// Mitsubishi GX Works2 project: plc_208837534_316493808   PLC: FX3G

// global labels: Global1
VAR_GLOBAL
  reset AT X010 : BOOL;
  EndDAY AT X005 : BOOL;
  cc17 AT CC17 : BOOL;
END_VAR
VAR_GLOBAL CONSTANT
  k_3 : INT := 3;
END_VAR
VAR_GLOBAL
  startDAY AT CS17 : BOOL;
  LAMP10 AT Y010 : BOOL;
  t_c_1 AT TC1 : BOOL;
END_VAR
VAR_GLOBAL CONSTANT
  k_5 : INT := 500;
END_VAR
VAR_GLOBAL
  LAMP11 AT Y011 : BOOL;
  m_0 AT M0 : BOOL;
END_VAR
VAR_GLOBAL CONSTANT
  k_1 : INT := 2000;
END_VAR
VAR_GLOBAL
  d_110 AT D1100 : INT;
  d_1110 AT D1110 : INT;
END_VAR
VAR_GLOBAL CONSTANT
  k_500 : INT := 50;
END_VAR
VAR_GLOBAL
  m_1 AT M1 : BOOL;
  t_c_3 AT TC3 : BOOL;
END_VAR
VAR_GLOBAL CONSTANT
  k_50 : INT := 50;
END_VAR
VAR_GLOBAL
  t_n_3 AT TN3 : INT;
  t_s_3 AT TS3 : BOOL;
END_VAR
VAR_GLOBAL CONSTANT
  Processing : REAL := 1350;
  Coating : REAL := 4500;
END_VAR
VAR_GLOBAL
  chocolate AT D1125 : REAL;
  StartOfProcessing AT X001 : BOOL;
  PeanutProcessing AT D1130 : REAL;
END_VAR
VAR_GLOBAL CONSTANT
  MAX150 : REAL := 150;
END_VAR
VAR_GLOBAL
  Peanut AT D1120 : REAL;
  HELP AT D1103 : INT;
  M_3 AT M3 : BOOL;
  m_4 AT M4 : BOOL;
  m_5 AT M5 : BOOL;
  LessThen70 AT M5 : BOOL;
  LessThen120 AT M6 : BOOL;
  LessThen150 AT M7 : BOOL;
END_VAR
VAR_GLOBAL CONSTANT
  k_120 : REAL := 120;
  k_150 : REAL := 150;
  k_70 : REAL := 70;
  k_20 : INT := 20;
  k_30 : INT := 30;
  k_40 : INT := 40;
END_VAR
VAR_GLOBAL
  m_8 AT M8 : BOOL;
  lampy1 AT Y001 : BOOL;
  d_1112 AT D1112 : INT;
  d_1114 AT D1114 : INT;
  d_1118 AT D1118 : INT;
  t_c_2 AT TC2 : BOOL;
  t_c_4 AT TC4 : BOOL;
  t_s_2 AT TS2 : BOOL;
  t_n_2 AT TN2 : INT;
  t_s_1 AT TS1 : BOOL;
  t_s_4 AT TS4 : BOOL;
  t_n_4 AT TN4 : INT;
END_VAR
VAR_GLOBAL CONSTANT
  k_45 : INT := 45;
  k_60 : INT := 60;
END_VAR
VAR_GLOBAL
  t_c_5 AT TC5 : BOOL;
  t_c_6 AT TC6 : BOOL;
  t_c_7 AT TC7 : BOOL;
  t_s_5 AT TS5 : BOOL;
  t_s_6 AT TS6 : BOOL;
  t_s_7 AT TS7 : BOOL;
  t_c_8 AT TC8 : BOOL;
  m_11 AT M11 : BOOL;
  t_s_8 AT TS8 : BOOL;
  t_c_9 AT TC9 : BOOL;
  t_s_9 AT TS9 : BOOL;
  LAMP3 AT Y003 : BOOL;
  t_c_10 AT TC10 : BOOL;
END_VAR
VAR_GLOBAL CONSTANT
  k_10 : INT := 10;
END_VAR
VAR_GLOBAL
  t_s_10 AT TS10 : BOOL;
  t_c_11 AT TC11 : BOOL;
  t_s_11 AT TS11 : BOOL;
  m_12 AT M12 : BOOL;
  t_n_10 AT TN10 : INT;
END_VAR
VAR_GLOBAL CONSTANT
  k_100 : INT := 100;
END_VAR
VAR_GLOBAL
  t_c_15 AT TC15 : BOOL;
  t_s_15 AT TS15 : BOOL;
  t_c_20 AT TC20 : BOOL;
  t_s_20 AT TS20 : BOOL;
  m_13 AT M13 : BOOL;
  t_c_25 AT TC25 : BOOL;
  t_s_25 AT TS25 : BOOL;
  t_n_25 AT TN25 : INT;
  t_n_15 AT TN15 : INT;
  d_1160 AT D1160 : INT;
  t_c_30 AT TC30 : BOOL;
  m_14 AT M14 : BOOL;
  t_s_30 AT TS30 : BOOL;
  m_15 AT M15 : BOOL;
  m_16 AT M16 : BOOL;
  m_17 AT M17 : BOOL;
END_VAR
VAR_GLOBAL CONSTANT
  MAX600chocolate : REAL := 600;
END_VAR
VAR_GLOBAL
  m_18 AT M18 : BOOL;
  readAnalog AT X007 : BOOL;
END_VAR
VAR_GLOBAL CONSTANT
  k_2_5 : REAL := 2.5;
  k_7 : REAL := 7;
END_VAR
VAR_GLOBAL
  m_19 AT M19 : BOOL;
END_VAR
VAR_GLOBAL CONSTANT
  k_9 : REAL := 9;
END_VAR
VAR_GLOBAL
  m_20 AT M20 : BOOL;
END_VAR
VAR_GLOBAL CONSTANT
  k_1_1 : REAL := 1;
END_VAR
VAR_GLOBAL
  m_21 AT M21 : BOOL;
  m_22 AT M22 : BOOL;
  m_23 AT M23 : BOOL;
  EndTransformationProcess AT M9 : BOOL;
  EndCuttingProcess AT M10 : BOOL;
END_VAR
VAR_GLOBAL CONSTANT
  k_0 : REAL;
END_VAR
VAR_GLOBAL
  analogIn2 AT D8281 : INT;
  valueBamba AT D1145 : REAL;
  d_1170 AT D1170 : INT;
END_VAR
VAR_GLOBAL CONSTANT
  K_397_2 : REAL := 397.2;
END_VAR
VAR_GLOBAL
  valueBambaGOOD AT D1150 : REAL;
  m_24 AT M24 : BOOL;
  EndValue AT M25 : BOOL;
END_VAR
VAR_GLOBAL CONSTANT
  k_1_5 : REAL := 1.5;
END_VAR
VAR_GLOBAL
  c_o AT M26 : BOOL;
  x_2 AT X002 : BOOL;
  x_3 AT X003 : BOOL;
  Coating_container AT D1135 : REAL;
  THERE_IS_CHOCOLATE AT M27 : BOOL;
  amountProsecs AT D1105 : REAL;
END_VAR
VAR_GLOBAL CONSTANT
  k_3_3 : REAL := 3;
END_VAR
VAR_GLOBAL
  m_28 AT M28 : BOOL;
  m_29 AT M29 : BOOL;
  time_Coating AT D1165 : INT;
END_VAR
VAR_GLOBAL CONSTANT
  k_4 : INT := 4;
  k_5_5 : INT := 50;
END_VAR
VAR_GLOBAL
  M_30 AT M30 : BOOL;
  t_c_40 AT TC40 : BOOL;
  t_s_40 AT TS40 : BOOL;
  t_c_45 AT TC45 : BOOL;
  t_s_45 AT TS45 : BOOL;
  y_6 AT Y006 : BOOL;
  t_c_50 AT TC50 : BOOL;
  t_s_50 AT TS50 : BOOL;
  M_31 AT M31 : BOOL;
END_VAR
VAR_GLOBAL CONSTANT
  k_2 : REAL := 2;
END_VAR
VAR_GLOBAL
  Bamba_bags AT D1175 : REAL;
  m_32 AT M32 : BOOL;
  Bamba_bags_int AT D1180 : INT;
  M_33 AT M33 : BOOL;
  M_34 AT M34 : BOOL;
  M_35 AT M35 : BOOL;
  M_36 AT M36 : BOOL;
END_VAR
VAR_GLOBAL CONSTANT
  k_50_0 : INT := 500;
END_VAR
VAR_GLOBAL
  M_37 AT M37 : BOOL;
END_VAR
VAR_GLOBAL CONSTANT
  k_5000 : INT := 5000;
END_VAR
VAR_GLOBAL
  M_38 AT M38 : BOOL;
  M_39 AT M39 : BOOL;
END_VAR
VAR_GLOBAL CONSTANT
  k_10_10 : INT := 10;
END_VAR
VAR_GLOBAL
  amout_Contenirs_to_int AT D1195 : INT;
  Bags AT D1185 : INT;
  Amount_Contenirs AT D1190 : INT;
  m_40 AT M40 : BOOL;
  modolu AT D1200 : INT;
  m_41 AT M41 : BOOL;
END_VAR
VAR_GLOBAL CONSTANT
  k_1_word : INT := 1;
END_VAR
VAR_GLOBAL
  m_42 AT M42 : BOOL;
END_VAR
VAR_GLOBAL CONSTANT
  k_0_0 : INT;
END_VAR
VAR_GLOBAL
  m_43 AT M43 : BOOL;
  Container_after_work_cot AT M44 : BOOL;
  Container_after_work_pean AT M45 : BOOL;
END_VAR
VAR_GLOBAL CONSTANT
  k_2500 : INT := 2500;
END_VAR
VAR_GLOBAL
  five_ton AT M46 : BOOL;
  t_c_70 AT TC70 : BOOL;
  t_s_70 AT TS70 : BOOL;
  lampy7 AT Y007 : BOOL;
  m_50 AT M50 : BOOL;
END_VAR
VAR_GLOBAL CONSTANT
  k_0_1 : REAL := 0.1;
END_VAR
VAR_GLOBAL
  there_is_peant AT M47 : BOOL;
  No_storage_space_END_DAY AT M49 : BOOL;
  Completion_coating_proces AT M51 : BOOL;
  Out_chocolate_stock AT M52 : BOOL;
  Out_peanut_stok AT M53 : BOOL;
  Conditions_ending_day AT M54 : BOOL;
END_VAR
VAR_GLOBAL CONSTANT
  k_2_WORD : INT := 2;
END_VAR
VAR_GLOBAL
  Duplication_performed AT M55 : BOOL;
END_VAR
VAR_GLOBAL CONSTANT
  k_1000 : REAL := 1000;
END_VAR
VAR_GLOBAL
  Distribution_made AT M56 : BOOL;
  Div_made AT M57 : BOOL;
  reset_variables AT M58 : BOOL;
END_VAR
VAR_GLOBAL CONSTANT
  K_397_2_WORD : INT := 397;
END_VAR
VAR_GLOBAL
  Several_processes AT CC20 : BOOL;
  cS20 AT CS20 : BOOL;
  bags_in_float AT D1240 : REAL;
  bamba_to_float AT M60 : BOOL;
  Amount_bamba_kg AT D1210 : REAL;
  Amount_bamba_ton AT D1220 : REAL;
  Amouny_bamba_analog AT D1230 : REAL;
  Bamab_output AT D1250 : INT;
  move_to_int AT M61 : BOOL;
  analog_output AT D8282 : INT;
  print_to_analog AT M62 : BOOL;
END_VAR
VAR_GLOBAL CONSTANT
  k_2_6 : REAL := 2.6;
  k_7_1 : REAL := 7.1;
  k_70_1 : REAL := 70.1;
  k_120_1 : REAL := 120.1;
END_VAR
VAR_GLOBAL
  M_63 AT M63 : BOOL;
END_VAR

// task Task_01 (event TRUE, interval 0, priority 31): POU_01

PROGRAM POU_01
(* structured ladder/FBD written out as ST: instructions are called as NAME(EN, inputs, outputs); _pN, _eN, _tN stand for wires *)
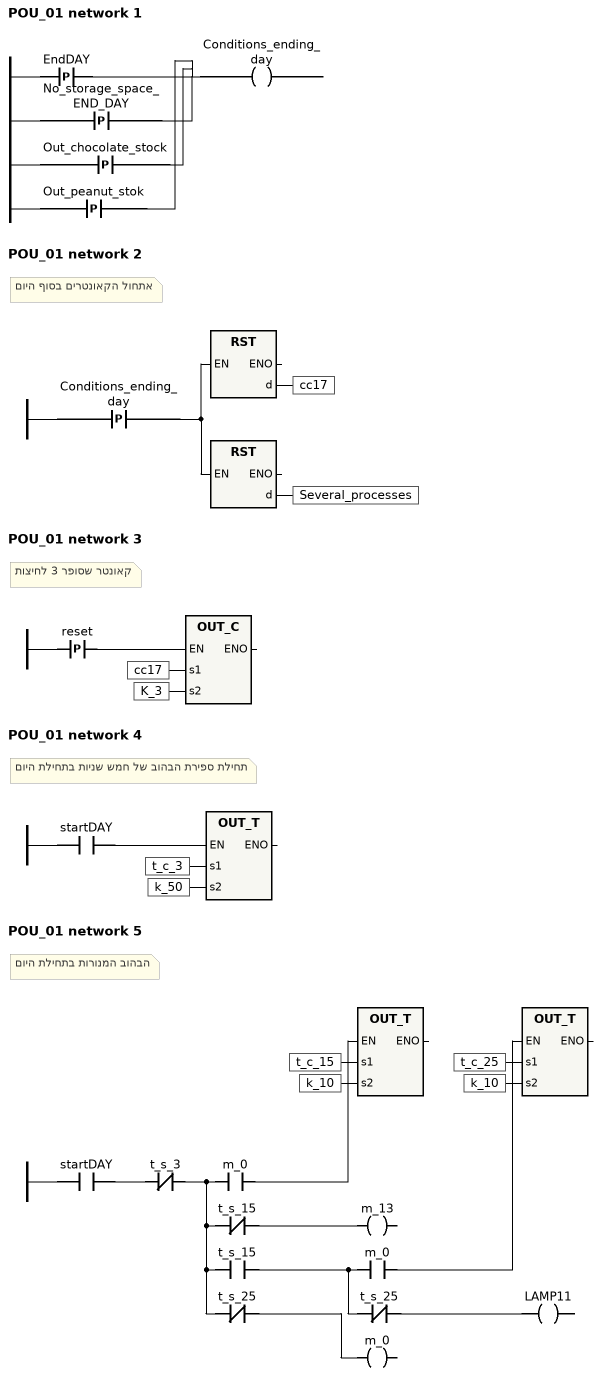
(* network 1 *)
Conditions_ending_day := LDP(TRUE, EndDAY) OR LDP(TRUE, No_storage_space_END_DAY) OR LDP(TRUE, Out_chocolate_stock) OR LDP(TRUE, Out_peanut_stok);
(* network 2 *)
(* אתחול הקאונטרים בסוף היום *)
_p1 := LDP(TRUE, Conditions_ending_day);
RST(_p1, cc17);
RST(_p1, Several_processes);
(* network 3 *)
(* קאונטר שסופר 3 לחיצות *)
OUT_C(LDP(TRUE, reset), cc17, K_3);
(* network 4 *)
(* תחילת ספירת הבהוב של חמש שניות בתחילת היום *)
OUT_T(startDAY, t_c_3, k_50);
(* network 5 *)
(* הבהוב המנורות בתחילת היום *)
_p1 := startDAY AND NOT t_s_3;
OUT_T(_p1 AND m_0, t_c_15, k_10);
m_13 := _p1 AND NOT t_s_15;
_p2 := _p1 AND t_s_15;
OUT_T(_p2 AND m_0, t_c_25, k_10);
LAMP11 := _p2 AND NOT t_s_25;
m_0 := _p1 AND NOT t_s_25;
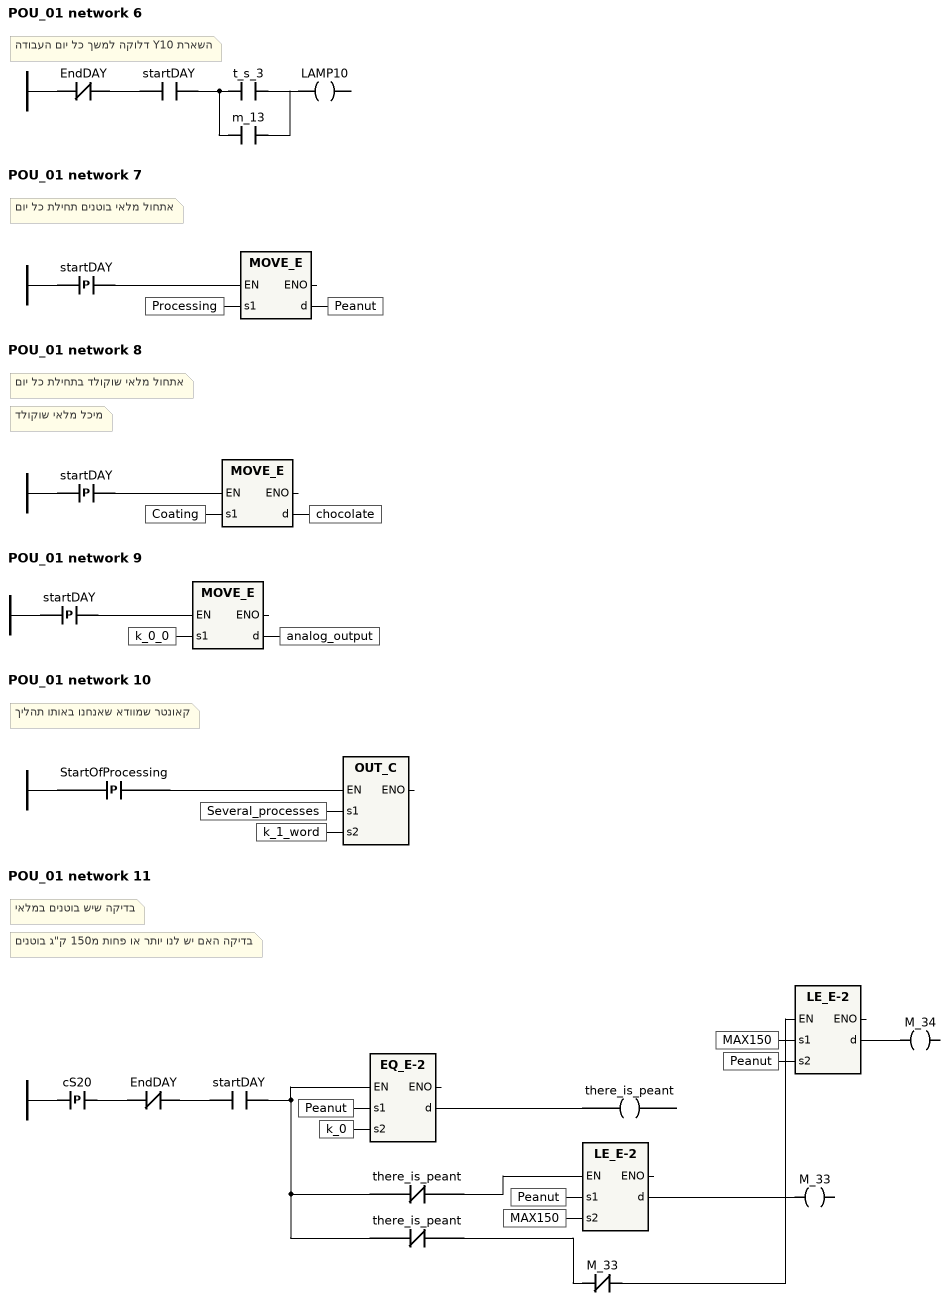
(* network 6 *)
(* השארת Y10 דלוקה למשך כל יום העבודה *)
_p1 := NOT EndDAY AND startDAY;
LAMP10 := (_p1 AND t_s_3) OR (_p1 AND m_13);
(* network 7 *)
(* אתחול מלאי בוטנים תחילת כל יום *)
MOVE_E(LDP(TRUE, startDAY), Processing, Peanut);
(* network 8 *)
(* אתחול מלאי שוקולד בתחילת כל יום *)
(* מיכל מלאי שוקולד *)
MOVE_E(LDP(TRUE, startDAY), Coating, chocolate);
(* network 9 *)
MOVE_E(LDP(TRUE, startDAY), k_0_0, analog_output);
(* network 10 *)
(* קאונטר שמוודא שאנחנו באותו תהליך *)
OUT_C(LDP(TRUE, StartOfProcessing), Several_processes, k_1_word);
(* network 11 *)
(* בדיקה שיש בוטנים במלאי *)
(* בדיקה האם יש לנו יותר או פחות מ150 ק"ג בוטנים *)
_p1 := LDP(TRUE, cS20) AND NOT EndDAY AND startDAY;
EQ_E(_p1, Peanut, k_0, _t2);
there_is_peant := _t2;
LE_E(_p1 AND NOT there_is_peant, Peanut, MAX150, _t3);
M_33 := _t3;
LE_E(_p1 AND NOT there_is_peant AND NOT M_33, MAX150, Peanut, _t4);
M_34 := _t4;
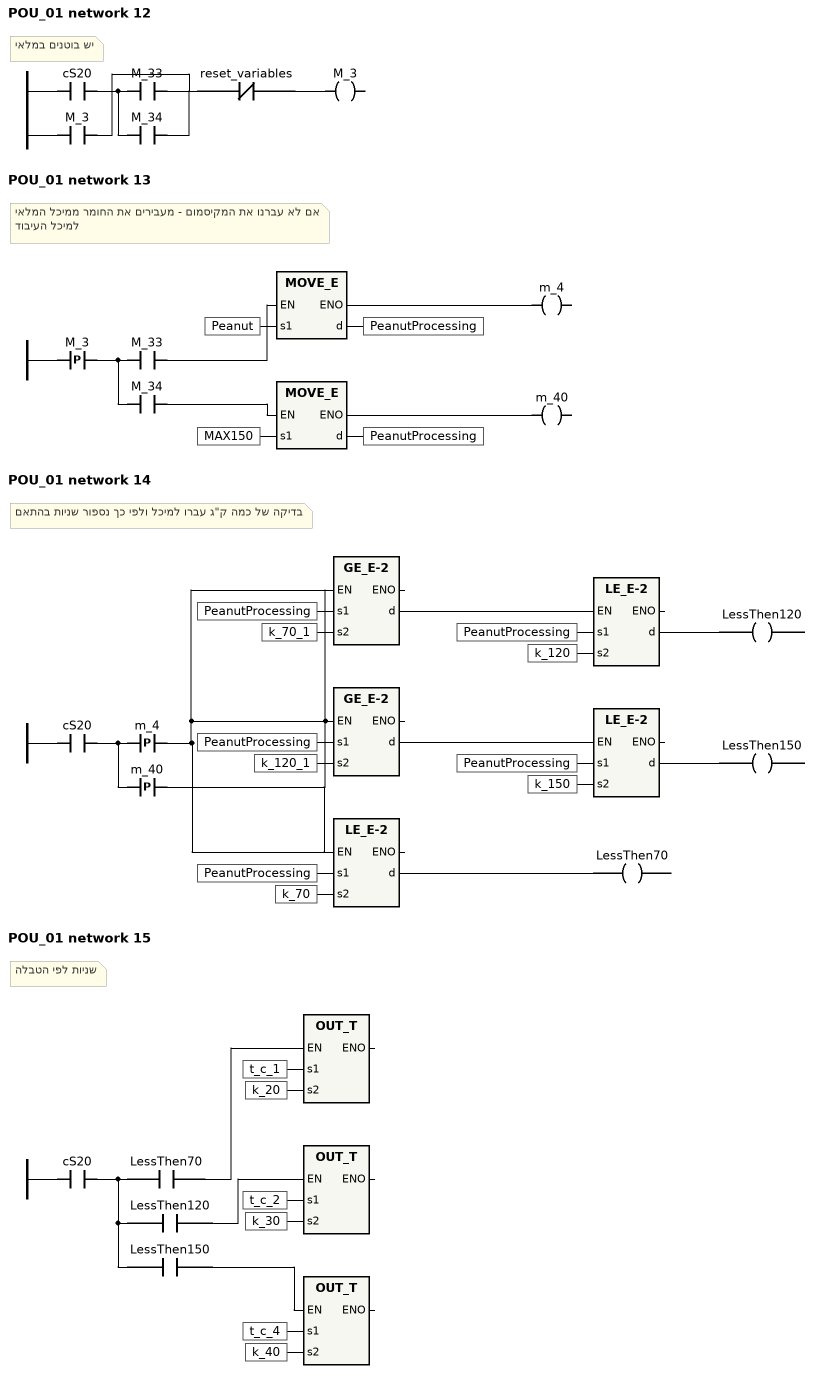
(* network 12 *)
(* יש בוטנים במלאי *)
M_3 := ((cS20 AND M_33) OR (cS20 AND M_34) OR M_3) AND NOT reset_variables;
(* network 13 *)
(* אם לא עברנו את המקיסמום - מעבירים את החומר ממיכל המלאי למיכל העיבוד *)
_p1 := LDP(TRUE, M_3);
_e2 := MOVE_E(_p1 AND M_33, Peanut, PeanutProcessing);
m_4 := _e2;
_e3 := MOVE_E(_p1 AND M_34, MAX150, PeanutProcessing);
m_40 := _e3;
(* network 14 *)
(* בדיקה של כמה ק"ג עברו למיכל ולפי כך נספור שניות בהתאם *)
_p1 := (cS20 AND LDP(TRUE, m_4)) OR (cS20 AND LDP(TRUE, m_40));
LE_E(_p1, PeanutProcessing, k_70, _t2);
LessThen70 := _t2;
GE_E(_p1, PeanutProcessing, k_70_1, _t3);
LE_E(_t3, PeanutProcessing, k_120, _t4);
LessThen120 := _t4;
GE_E(_p1, PeanutProcessing, k_120_1, _t5);
LE_E(_t5, PeanutProcessing, k_150, _t6);
LessThen150 := _t6;
(* network 15 *)
(* שניות לפי הטבלה *)
OUT_T(cS20 AND LessThen70, t_c_1, k_20);
OUT_T(cS20 AND LessThen120, t_c_2, k_30);
OUT_T(cS20 AND LessThen150, t_c_4, k_40);
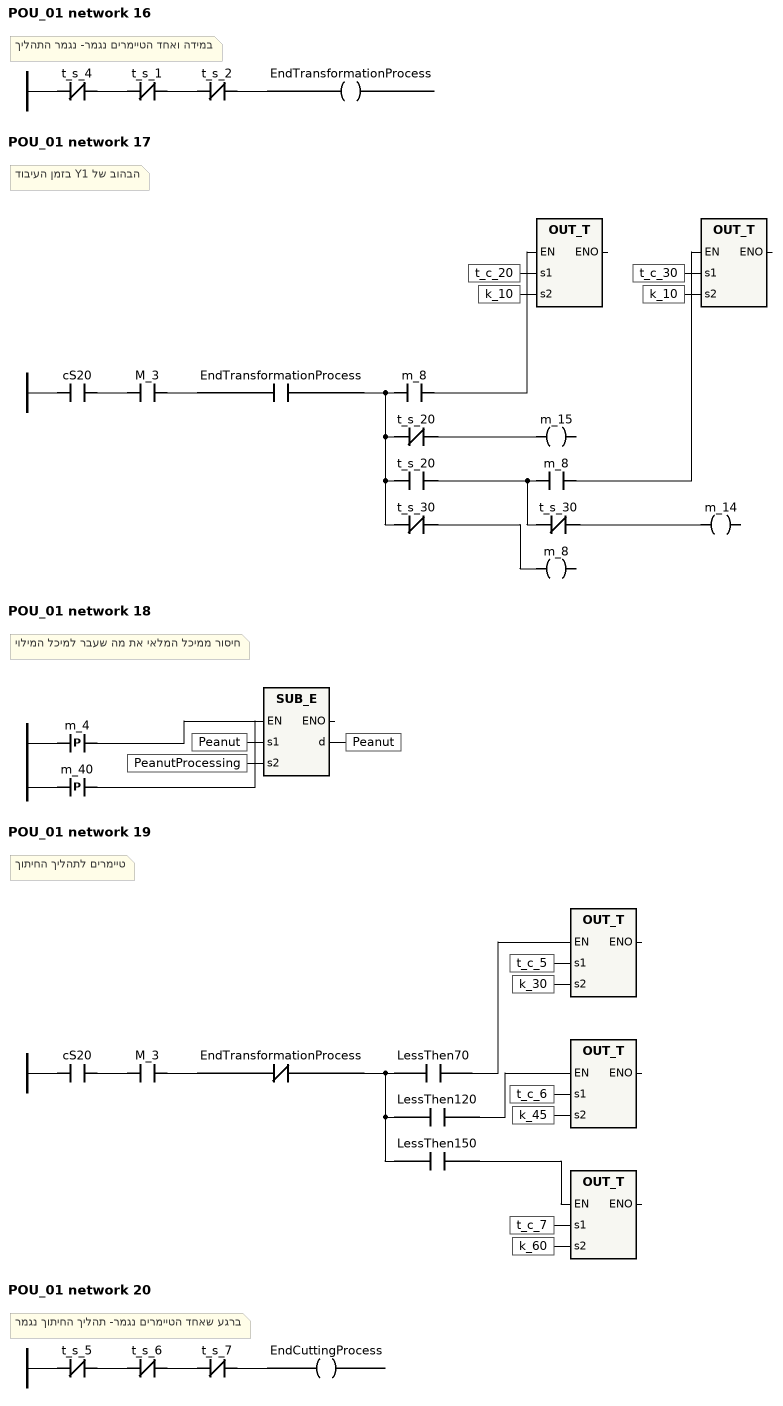
(* network 16 *)
(* במידה ואחד הטיימרים נגמר- נגמר התהליך *)
EndTransformationProcess := NOT t_s_4 AND NOT t_s_1 AND NOT t_s_2;
(* network 17 *)
(* הבהוב של Y1 בזמן העיבוד *)
_p1 := cS20 AND M_3 AND EndTransformationProcess;
OUT_T(_p1 AND m_8, t_c_20, k_10);
m_15 := _p1 AND NOT t_s_20;
_p2 := _p1 AND t_s_20;
OUT_T(_p2 AND m_8, t_c_30, k_10);
m_14 := _p2 AND NOT t_s_30;
m_8 := _p1 AND NOT t_s_30;
(* network 18 *)
(* חיסור ממיכל המלאי את מה שעבר למיכל המילוי *)
SUB_E(LDP(TRUE, m_4) OR LDP(TRUE, m_40), Peanut, PeanutProcessing, Peanut);
(* network 19 *)
(* טיימרים לתהליך החיתוך *)
_p1 := cS20 AND M_3 AND NOT EndTransformationProcess;
OUT_T(_p1 AND LessThen70, t_c_5, k_30);
OUT_T(_p1 AND LessThen120, t_c_6, k_45);
OUT_T(_p1 AND LessThen150, t_c_7, k_60);
(* network 20 *)
(* ברגע שאחד הטיימרים נגמר- תהליך החיתוך נגמר *)
EndCuttingProcess := NOT t_s_5 AND NOT t_s_6 AND NOT t_s_7;
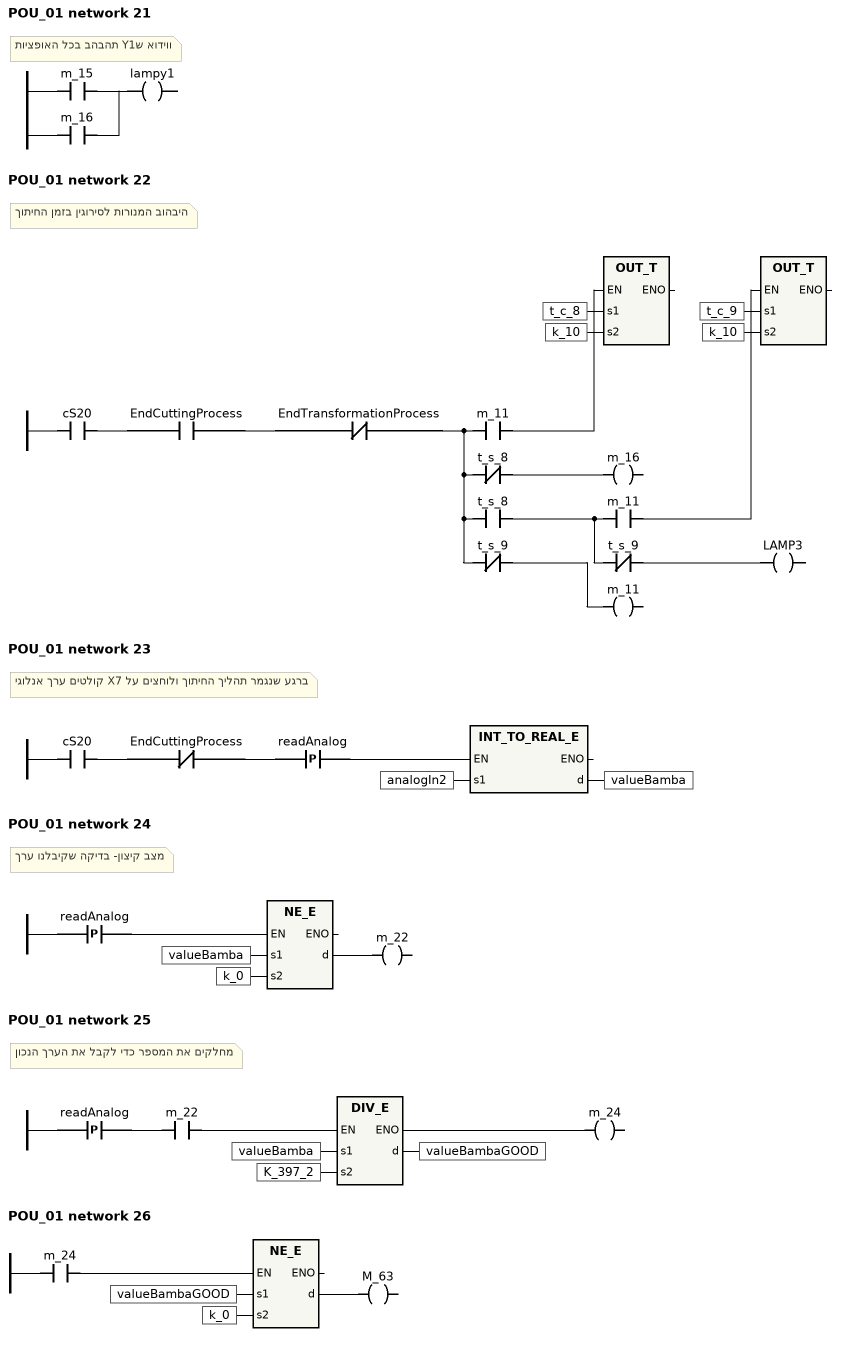
(* network 21 *)
(* ווידוא שY1 תהבהב בכל האופציות *)
lampy1 := m_15 OR m_16;
(* network 22 *)
(* היבהוב המנורות לסירוגין בזמן החיתוך *)
_p1 := cS20 AND EndCuttingProcess AND NOT EndTransformationProcess;
OUT_T(_p1 AND m_11, t_c_8, k_10);
m_16 := _p1 AND NOT t_s_8;
_p2 := _p1 AND t_s_8;
OUT_T(_p2 AND m_11, t_c_9, k_10);
LAMP3 := _p2 AND NOT t_s_9;
m_11 := _p1 AND NOT t_s_9;
(* network 23 *)
(* ברגע שנגמר תהליך החיתוך ולוחצים על X7 קולטים ערך אנלוגי *)
INT_TO_REAL_E(cS20 AND NOT EndCuttingProcess AND LDP(TRUE, readAnalog), analogIn2, valueBamba);
(* network 24 *)
(* מצב קיצון- בדיקה שקיבלנו ערך *)
NE_E(LDP(TRUE, readAnalog), valueBamba, k_0, _t1);
m_22 := _t1;
(* network 25 *)
(* מחלקים את המספר כדי לקבל את הערך הנכון *)
_e1 := DIV_E(LDP(TRUE, readAnalog) AND m_22, valueBamba, K_397_2, valueBambaGOOD);
m_24 := _e1;
(* network 26 *)
NE_E(m_24, valueBambaGOOD, k_0, _t1);
M_63 := _t1;
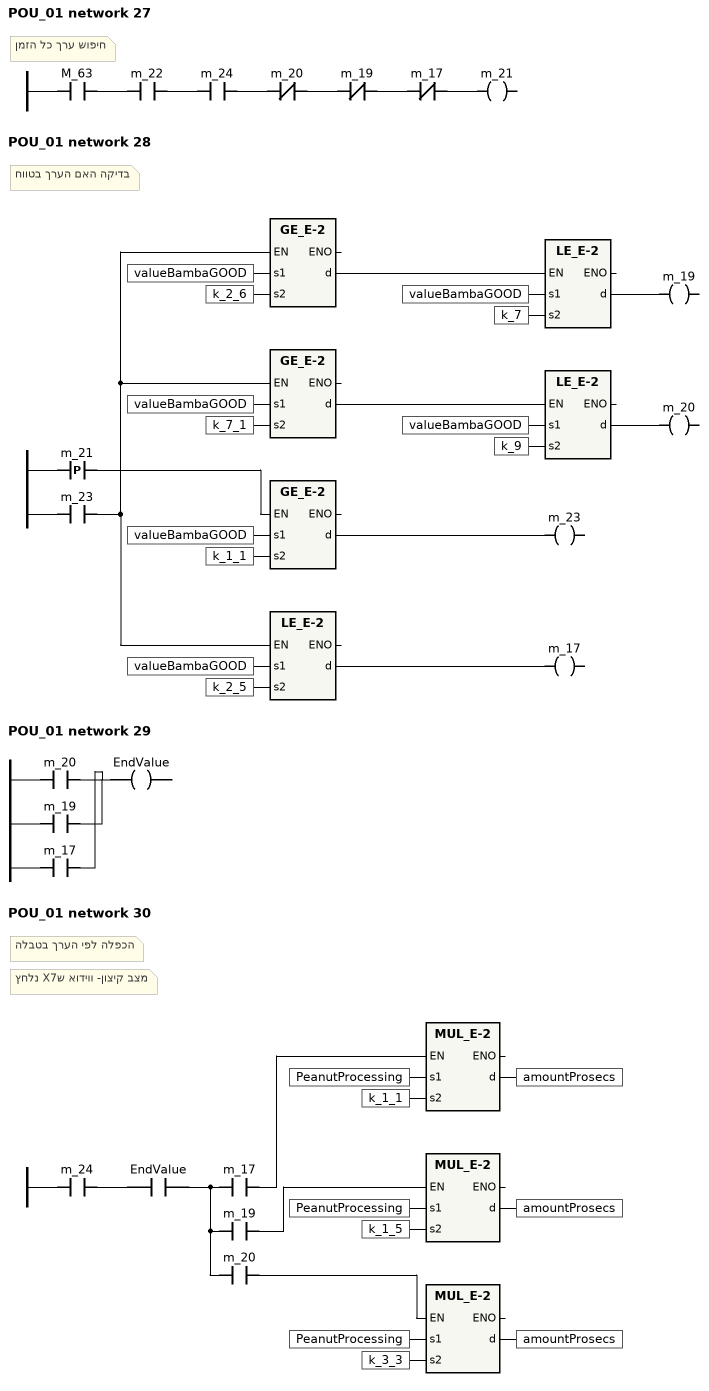
(* network 27 *)
(* חיפוש ערך כל הזמן *)
m_21 := M_63 AND m_22 AND m_24 AND NOT m_20 AND NOT m_19 AND NOT m_17;
(* network 28 *)
(* בדיקה האם הערך בטווח *)
GE_E(LDP(TRUE, m_21), valueBambaGOOD, k_1_1, _t1);
m_23 := _t1;
LE_E(m_23, valueBambaGOOD, k_2_5, _t2);
m_17 := _t2;
GE_E(m_23, valueBambaGOOD, k_2_6, _t3);
LE_E(_t3, valueBambaGOOD, k_7, _t4);
m_19 := _t4;
GE_E(m_23, valueBambaGOOD, k_7_1, _t5);
LE_E(_t5, valueBambaGOOD, k_9, _t6);
m_20 := _t6;
(* network 29 *)
EndValue := m_20 OR m_19 OR m_17;
(* network 30 *)
(* הכפלה לפי הערך בטבלה *)
(* מצב קיצון- ווידוא שX7 נלחץ *)
_p1 := m_24 AND EndValue;
MUL_E(_p1 AND m_17, PeanutProcessing, k_1_1, amountProsecs);
MUL_E(_p1 AND m_19, PeanutProcessing, k_1_5, amountProsecs);
MUL_E(_p1 AND m_20, PeanutProcessing, k_3_3, amountProsecs);
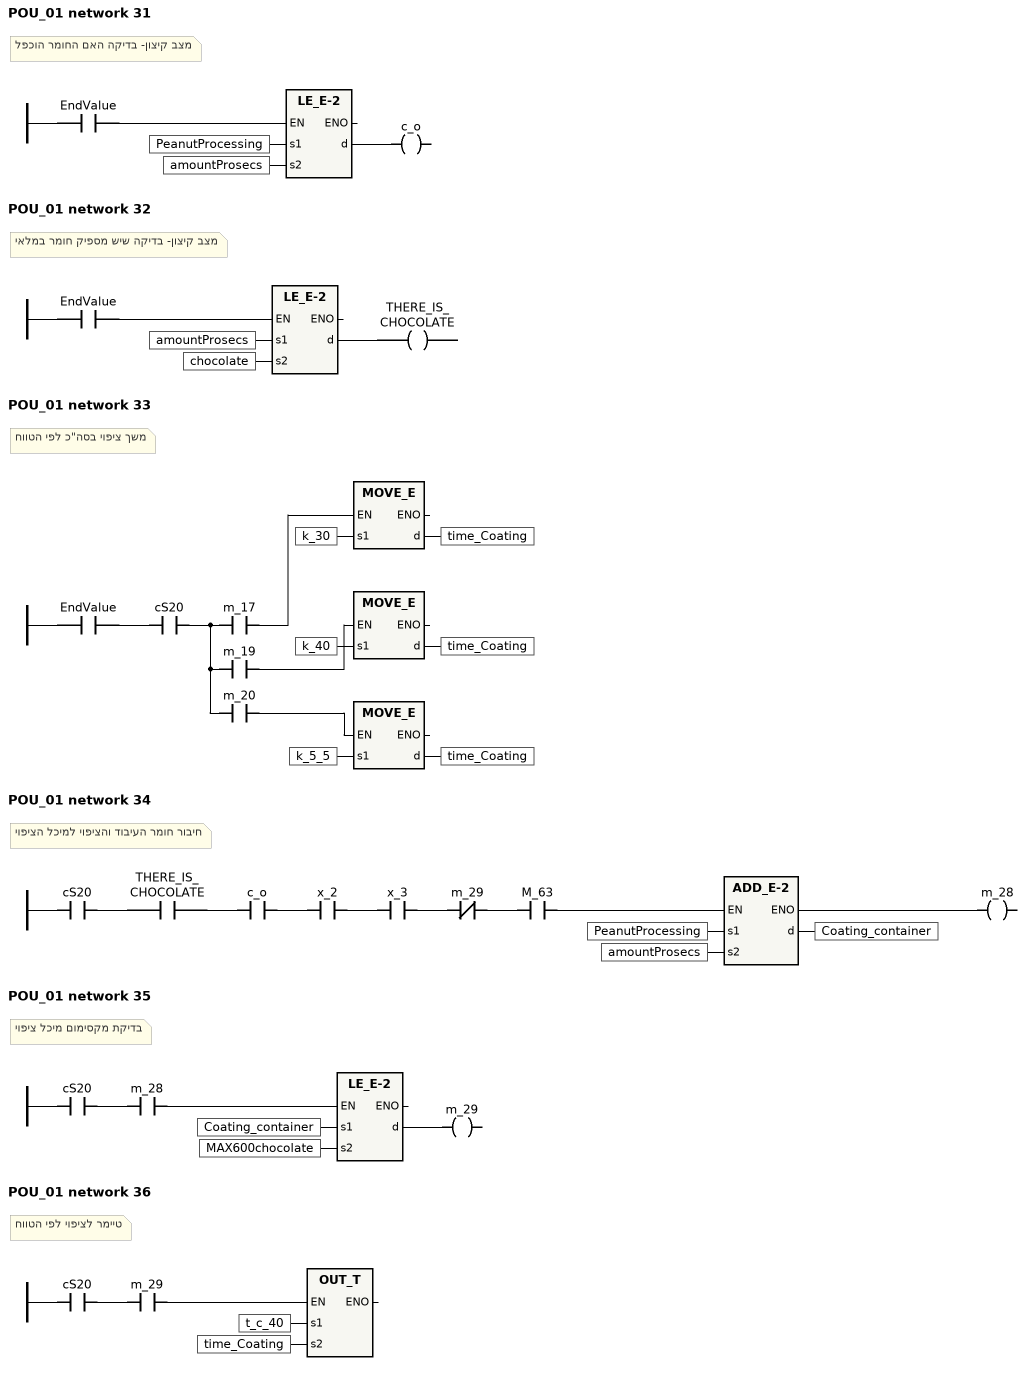
(* network 31 *)
(* מצב קיצון- בדיקה האם החומר הוכפל *)
LE_E(EndValue, PeanutProcessing, amountProsecs, _t1);
c_o := _t1;
(* network 32 *)
(* מצב קיצון- בדיקה שיש מספיק חומר במלאי *)
LE_E(EndValue, amountProsecs, chocolate, _t1);
THERE_IS_CHOCOLATE := _t1;
(* network 33 *)
(* משך ציפוי בסה"כ לפי הטווח *)
_p1 := EndValue AND cS20;
MOVE_E(_p1 AND m_17, k_30, time_Coating);
MOVE_E(_p1 AND m_19, k_40, time_Coating);
MOVE_E(_p1 AND m_20, k_5_5, time_Coating);
(* network 34 *)
(* חיבור חומר העיבוד והציפוי למיכל הציפוי *)
_e1 := ADD_E(cS20 AND THERE_IS_CHOCOLATE AND c_o AND x_2 AND x_3 AND NOT m_29 AND M_63, PeanutProcessing, amountProsecs, Coating_container);
m_28 := _e1;
(* network 35 *)
(* בדיקת מקסימום מיכל ציפוי *)
LE_E(cS20 AND m_28, Coating_container, MAX600chocolate, _t1);
m_29 := _t1;
(* network 36 *)
(* טיימר לציפוי לפי הטווח *)
OUT_T(cS20 AND m_29, t_c_40, time_Coating);
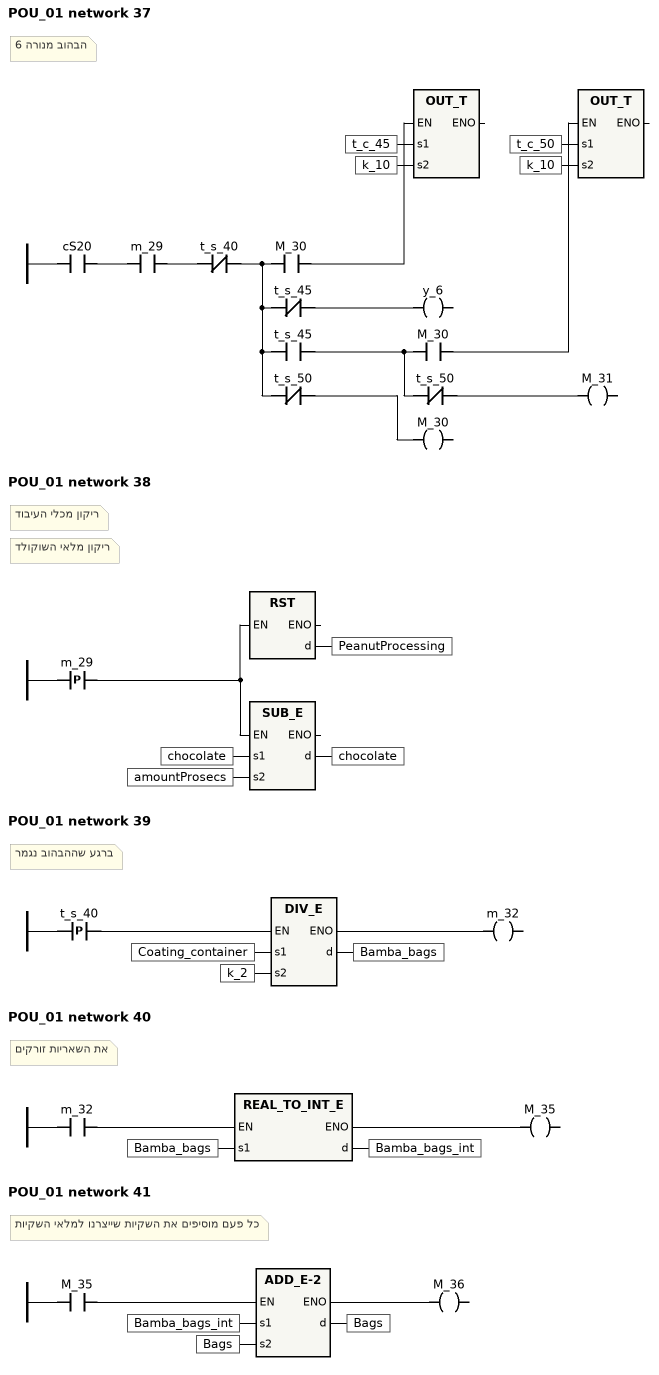
(* network 37 *)
(* הבהוב מנורה 6 *)
_p1 := cS20 AND m_29 AND NOT t_s_40;
OUT_T(_p1 AND M_30, t_c_45, k_10);
y_6 := _p1 AND NOT t_s_45;
_p2 := _p1 AND t_s_45;
OUT_T(_p2 AND M_30, t_c_50, k_10);
M_31 := _p2 AND NOT t_s_50;
M_30 := _p1 AND NOT t_s_50;
(* network 38 *)
(* ריקון מכלי העיבוד *)
(* ריקון מלאי השוקולד *)
_p1 := LDP(TRUE, m_29);
RST(_p1, PeanutProcessing);
SUB_E(_p1, chocolate, amountProsecs, chocolate);
(* network 39 *)
(* ברגע שההבהוב נגמר *)
_e1 := DIV_E(LDP(TRUE, t_s_40), Coating_container, k_2, Bamba_bags);
m_32 := _e1;
(* network 40 *)
(* את השאריות זורקים *)
_e1 := REAL_TO_INT_E(m_32, Bamba_bags, Bamba_bags_int);
M_35 := _e1;
(* network 41 *)
(* כל פעם מוסיפים את השקיות שייצרנו למלאי השקיות *)
_e1 := ADD_E(M_35, Bamba_bags_int, Bags, Bags);
M_36 := _e1;
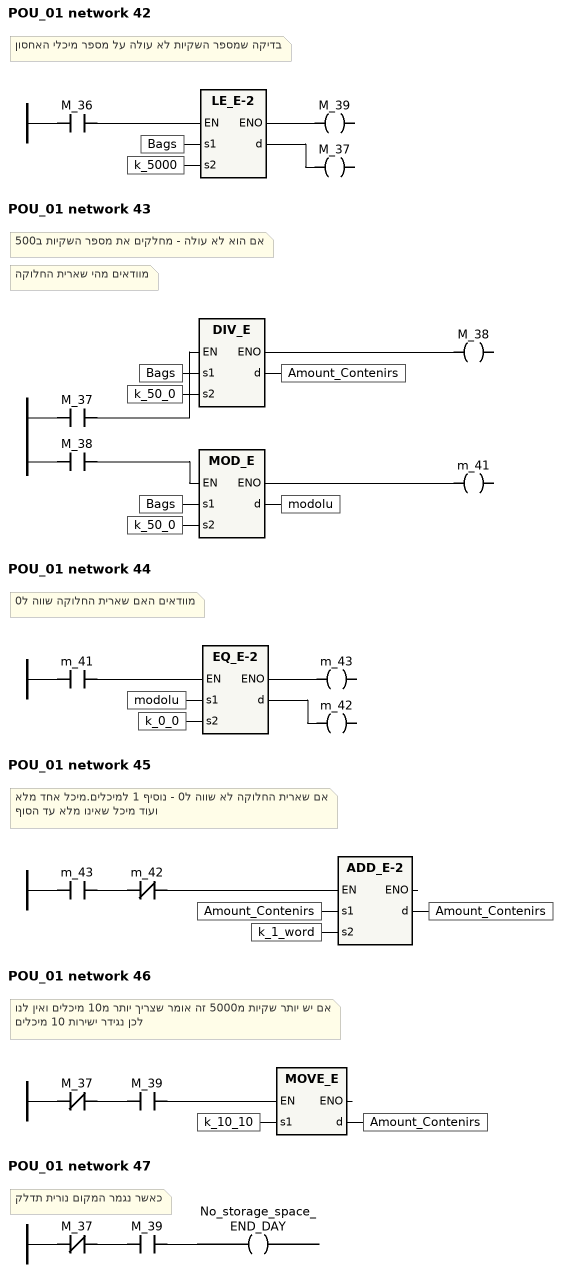
(* network 42 *)
(* בדיקה שמספר השקיות לא עולה על מספר מיכלי האחסון *)
_e2 := LE_E(M_36, Bags, k_5000, _t1);
M_39 := _e2;
M_37 := _t1;
(* network 43 *)
(* אם הוא לא עולה - מחלקים את מספר השקיות ב500 *)
(* מוודאים מהי שארית החלוקה *)
_e1 := DIV_E(M_37, Bags, k_50_0, Amount_Contenirs);
M_38 := _e1;
_e2 := MOD_E(M_38, Bags, k_50_0, modolu);
m_41 := _e2;
(* network 44 *)
(* מוודאים האם שארית החלוקה שווה ל0 *)
_e2 := EQ_E(m_41, modolu, k_0_0, _t1);
m_43 := _e2;
m_42 := _t1;
(* network 45 *)
(* אם שארית החלוקה לא שווה ל0 - נוסיף 1 למיכלים.מיכל אחד מלא ועוד מיכל שאינו מלא עד הסוף *)
ADD_E(m_43 AND NOT m_42, Amount_Contenirs, k_1_word, Amount_Contenirs);
(* network 46 *)
(* אם יש יותר שקיות מ5000 זה אומר שצריך יותר מ10 מיכלים ואין לנו לכן נגידר ישירות 10 מיכלים *)
MOVE_E(NOT M_37 AND M_39, k_10_10, Amount_Contenirs);
(* network 47 *)
(* כאשר נגמר המקום נורית תדלק *)
No_storage_space_END_DAY := NOT M_37 AND M_39;
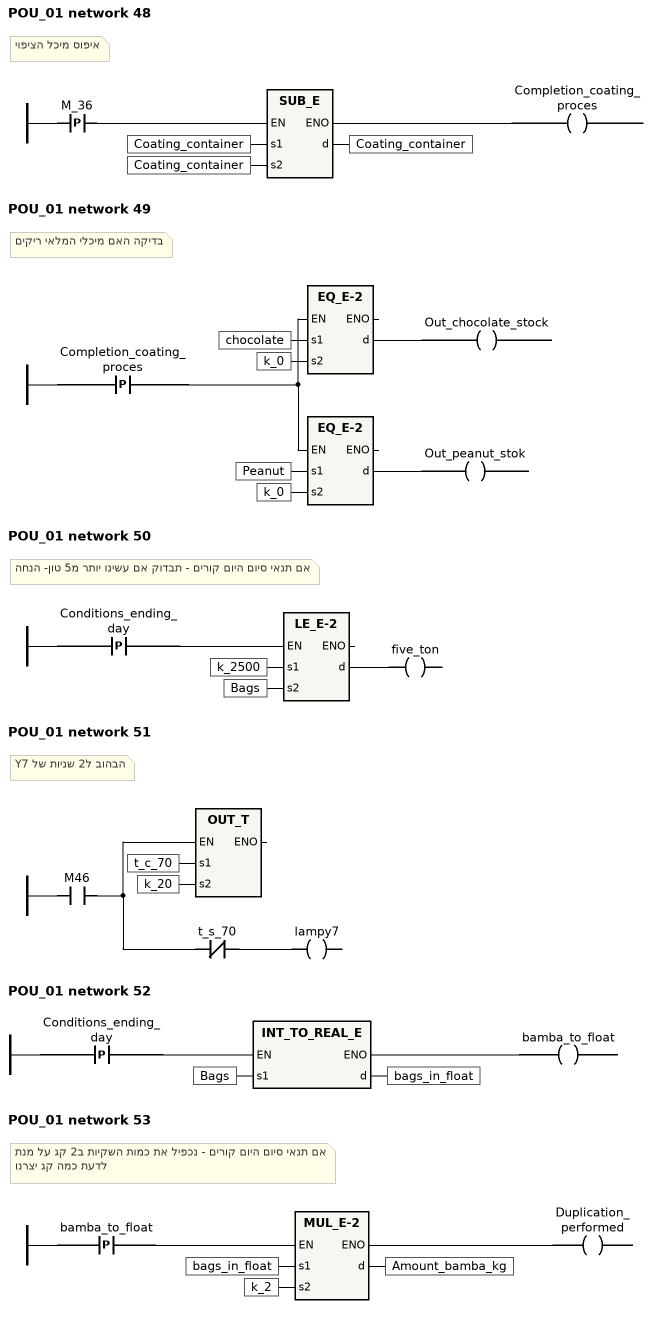
(* network 48 *)
(* איפוס מיכל הציפוי *)
_e1 := SUB_E(LDP(TRUE, M_36), Coating_container, Coating_container, Coating_container);
Completion_coating_proces := _e1;
(* network 49 *)
(* בדיקה האם מיכלי המלאי ריקים *)
_p1 := LDP(TRUE, Completion_coating_proces);
EQ_E(_p1, chocolate, k_0, _t2);
Out_chocolate_stock := _t2;
EQ_E(_p1, Peanut, k_0, _t3);
Out_peanut_stok := _t3;
(* network 50 *)
(* אם תנאי סיום היום קורים - תבדוק אם עשינו יותר מ5 טון- הנחה *)
LE_E(LDP(TRUE, Conditions_ending_day), k_2500, Bags, _t1);
five_ton := _t1;
(* network 51 *)
(* הבהוב ל2 שניות של Y7 *)
OUT_T(M46, t_c_70, k_20);
lampy7 := M46 AND NOT t_s_70;
(* network 52 *)
_e1 := INT_TO_REAL_E(LDP(TRUE, Conditions_ending_day), Bags, bags_in_float);
bamba_to_float := _e1;
(* network 53 *)
(* אם תנאי סיום היום קורים - נכפיל את כמות השקיות ב2 קג על מנת לדעת כמה קג יצרנו *)
_e1 := MUL_E(LDP(TRUE, bamba_to_float), bags_in_float, k_2, Amount_bamba_kg);
Duplication_performed := _e1;
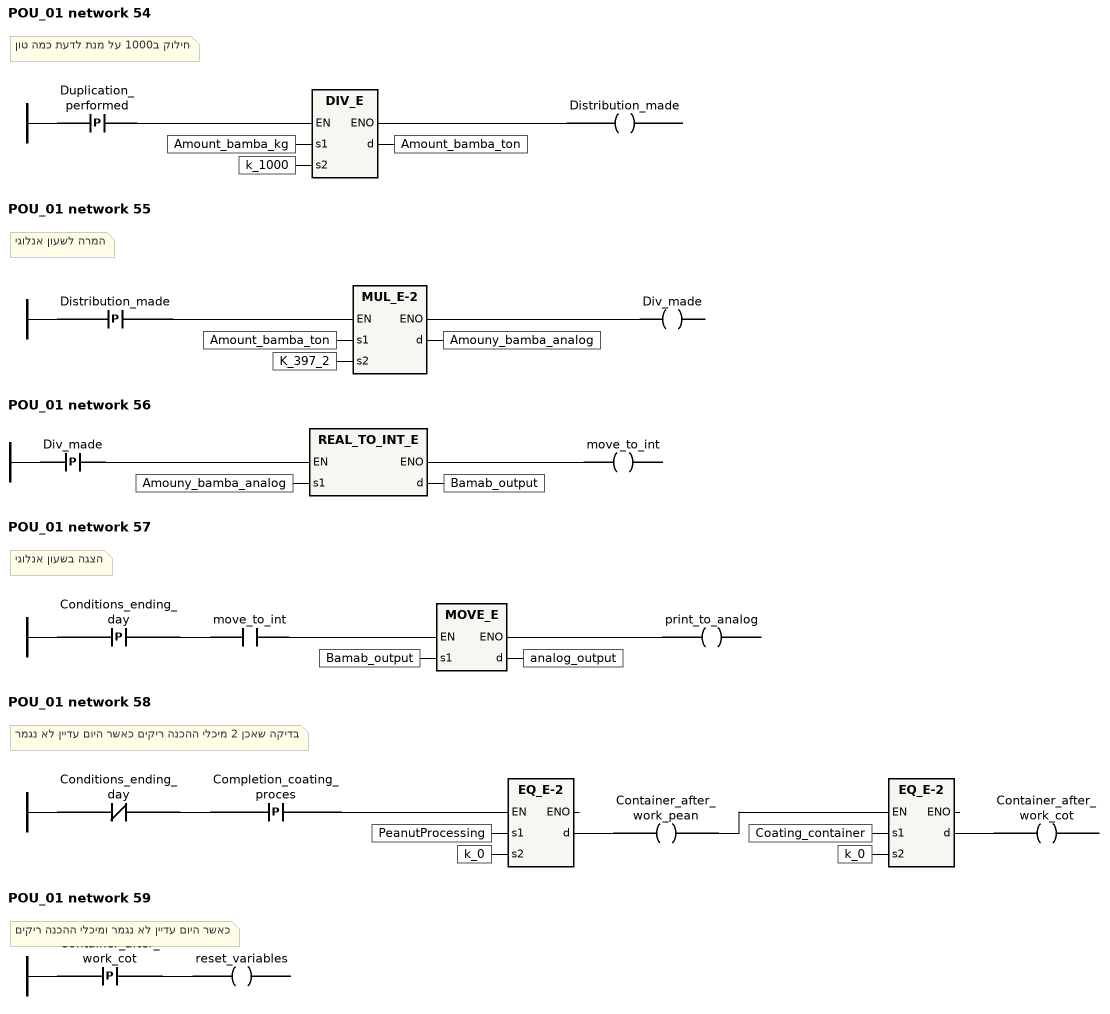
(* network 54 *)
(* חילוק ב1000 על מנת לדעת כמה טון *)
_e1 := DIV_E(LDP(TRUE, Duplication_performed), Amount_bamba_kg, k_1000, Amount_bamba_ton);
Distribution_made := _e1;
(* network 55 *)
(* המרה לשעון אנלוגי *)
_e1 := MUL_E(LDP(TRUE, Distribution_made), Amount_bamba_ton, K_397_2, Amouny_bamba_analog);
Div_made := _e1;
(* network 56 *)
_e1 := REAL_TO_INT_E(LDP(TRUE, Div_made), Amouny_bamba_analog, Bamab_output);
move_to_int := _e1;
(* network 57 *)
(* הצגה בשעון אנלוגי *)
_e1 := MOVE_E(LDP(TRUE, Conditions_ending_day) AND move_to_int, Bamab_output, analog_output);
print_to_analog := _e1;
(* network 58 *)
(* בדיקה שאכן 2 מיכלי ההכנה ריקים כאשר היום עדיין לא נגמר *)
EQ_E(NOT Conditions_ending_day AND LDP(TRUE, Completion_coating_proces), PeanutProcessing, k_0, _t1);
Container_after_work_pean := _t1;
EQ_E(_t1, Coating_container, k_0, _t2);
Container_after_work_cot := _t2;
(* network 59 *)
(* כאשר היום עדיין לא נגמר ומיכלי ההכנה ריקים *)
reset_variables := LDP(TRUE, Container_after_work_cot);
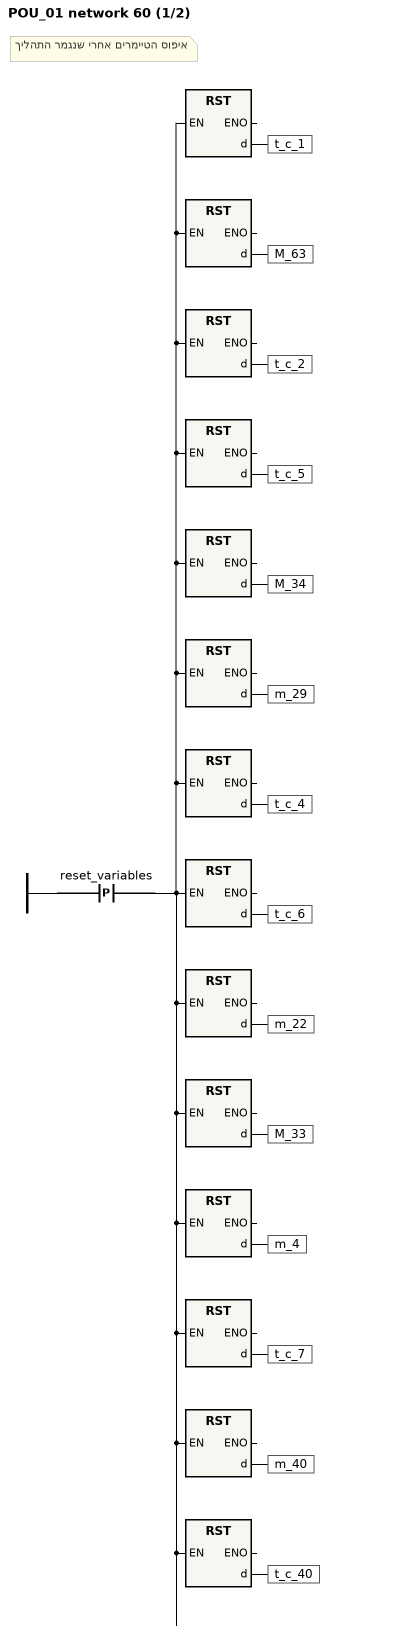
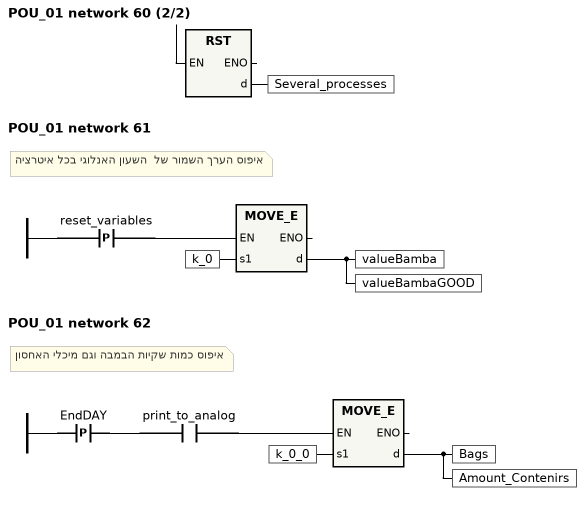
(* network 60 *)
(* איפוס הטיימרים אחרי שנגמר התהליך *)
_p1 := LDP(TRUE, reset_variables);
RST(_p1, t_c_1);
RST(_p1, t_c_2);
RST(_p1, M_63);
RST(_p1, t_c_5);
RST(_p1, M_34);
RST(_p1, m_29);
RST(_p1, t_c_4);
RST(_p1, t_c_6);
RST(_p1, m_22);
RST(_p1, t_c_7);
RST(_p1, M_33);
RST(_p1, m_4);
RST(_p1, m_40);
RST(_p1, t_c_40);
RST(_p1, Several_processes);
(* network 61 *)
(* איפוס הערך השמור של  השעון האנלוגי בכל איטרציה *)
MOVE_E(LDP(TRUE, reset_variables), k_0, valueBamba);
valueBambaGOOD := valueBamba;
(* network 62 *)
(* איפוס כמות שקיות הבמבה וגם מיכלי האחסון *)
MOVE_E(LDP(TRUE, EndDAY) AND print_to_analog, k_0_0, Bags);
Amount_Contenirs := Bags;
END_PROGRAM
